/// Update the variable display value in the Numpad for hex or dec and change the radio button.
/// This function is an enhancement of function VisuDlg_CheckedChangeNumberFormat, that also modifies
/// the caret and selection if the caret would be outside the text after the change of the display format.
/// :return: Not used, always FALSE
FUNCTION VisuDlg_ProcessChangeNumberFormat : BOOL
VAR_IN_OUT
	stOutputValue : STRING;
	stVariableValue : STRING;
	stMin : STRING;
	stMax : STRING;
	iFormatValue : INT;
	/// The current position of the caret. Either within the text or at the end of the text
	iCaretPosition	: INT;
	/// The start of the selected text (1-relative)
	iSelectionStart	: INT;
	/// The end of the selected text (1-relative).
	iSelectionEnd	: INT;
END_VAR
VAR_INPUT
	bPassword: BOOL;
	// use this way, because of integrated visu
	// 0. dec , 1. hex
	stClickedRadio : STRING;
END_VAR
VAR
	i : INT;	
	bChanged : BOOL;
	iTextLengthBeforeChange	: INT;
END_VAR

// simulate the radio button change
IF iFormatValue = Dialog_FormatTypes.HEX AND stClickedRadio = '0' THEN
	iFormatValue := Dialog_FormatTypes.DECIMAL;	
	bChanged := TRUE;
ELSIF iFormatValue = Dialog_FormatTypes.DECIMAL AND stClickedRadio = '1' THEN
	iFormatValue := Dialog_FormatTypes.HEX;
	bChanged := TRUE;
END_IF

// do some additional stuff
IF bChanged THEN
	// In order to check, whether the caret and/or selection has to be adjusted, we determine
	// the text length before the change, that corresponds to the parameters iCaretPosition and iSelection[Start|End]
	iTextLengthBeforeChange := LEN(stVariableValue);

	IF iFormatValue = Dialog_FormatTypes.HEX THEN	
		IF g_XExp THEN
			// first change the value to float:
			VisuDlg_CheckedExpFloatFormatSwitch(stOutputValue, stVariableValue, bPassword);
		END_IF
		stVariableValue := VisuDlgUtil_FormatValueToHex(stVariableValue);
		
		IF stMin <> '' THEN
			stMin := VisuDlgUtil_FormatExpToG(stMin);
		END_IF
		IF stMax <> '' THEN
			stMax := VisuDlgUtil_FormatExpToG(stMax);
		END_IF
	ELSE	
		stVariableValue := VisuDlgUtil_FormatValueToDec(stVariableValue);
		IF stMin <> '' THEN
			stMin := VisuDlgUtil_FormatValueToDec(stMin);
		END_IF
		IF stMax <> '' THEN
			stMax := VisuDlgUtil_FormatValueToDec(stMax);
		END_IF
	END_IF
	
	VisuDlgUtil_UpdateOutputValue(stOutputValue, stVariableValue, bPassword);
	
	// We adjust the caret and the selection.
	VisuDlgUtil_AdjustCaretAndSelectionAfterNumberFormatChange(
		iTextLengthBeforeChange,
		stVariableValue,
		iCaretPosition,
		iSelectionStart,
		iSelectionEnd
	);
END_IF

END_FUNCTION

(* stored: Version 1.1.0.1, ProductVersion 3.1.4024.2
   POU VisuDlg_ProcessChangeNumberFormat: Id {c57df06d-08fc-4e80-99c2-504d48246d54}, SpecialFunc None *)
